// Mitsubishi GX Works2 project: 折管检查机源程序   PLC: FX3S

PROGRAM MAIN
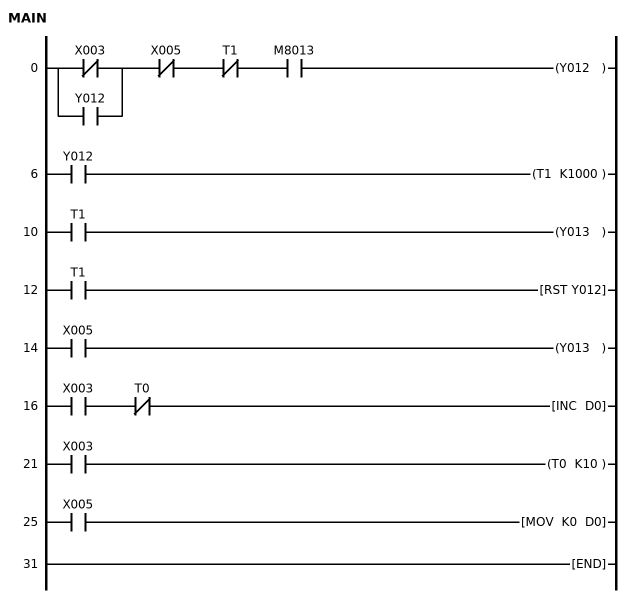
0     LDI     X003
      OR      Y012
      ANI     X005
      ANI     T1
      AND     M8013
      OUT     Y012
6     LD      Y012
      OUT     T1 K1000
10    LD      T1
      OUT     Y013
12    LD      T1
      RST     Y012
14    LD      X005
      OUT     Y013
16    LD      X003
      ANI     T0
      INC     D0
21    LD      X003
      OUT     T0 K10
25    LD      X005
      MOV     K0 D0
31    END
END_PROGRAM
